KUKA KRL program: dockof_2.src, dockof_2.dat

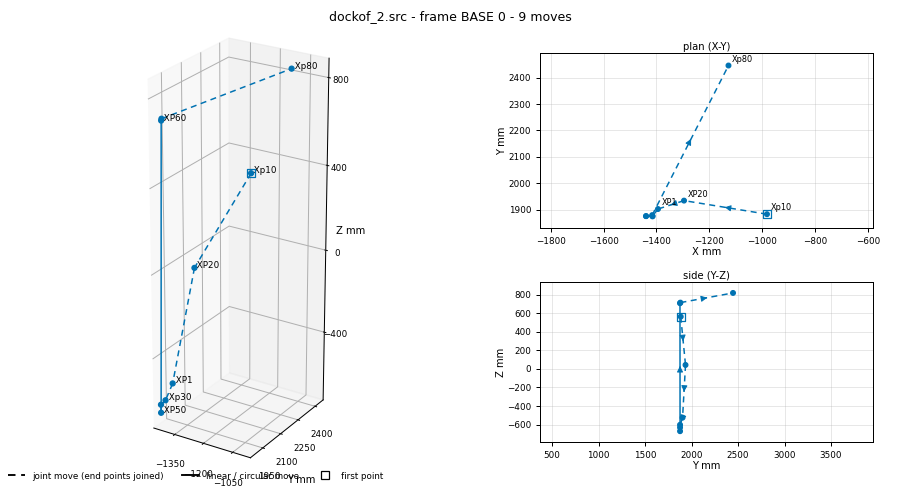
[picture p0: tool path of dockof_2.src in frame BASE 0, 9 of 9 moves have a stored position in this frame; points joined in program order, loops and branches not executed]
--- dockof_2.src ---
&ACCESS RV1
&REL 140
&COMMENT PLACE GUN 2
DEF DOCKOF_2( )
;================================================
; MODEL    :
; IE GROUP :
; STATION  :
; ROBOT    :
; FUNCTION : DOCK OFF GUN 2
;================================================
;FOLD INI
;FOLD BASISTECH INI
GLOBAL INTERRUPT DECL 3 WHEN $STOPMESS==TRUE DO IR_STOPM ( )
INTERRUPT ON 3
BAS (#INITMOV,0 )
;ENDFOLD (BASISTECH INI)
;FOLD GRIPPERTECH INI
USER_GRP(0,DUMMY,DUMMY,GDEFAULT)
;ENDFOLD (GRIPPERTECH INI)
;FOLD USER INI
;Make your modifications here

;ENDFOLD (USER INI)
;ENDFOLD (INI)

;FOLD PTP p10  Vel= 100 % H Tool[2]:Gun2 Base[0];%{PE}%R 5.4.35,%MKUKATPBASIS,%CMOVE,%VPTP,%P 1:PTP, 2:p10, 3:, 5:100, 7:H
$BWDSTART=FALSE
PDAT_ACT=PH
FDAT_ACT=Fp10
BAS(#PTP_PARAMS,100)
PTP Xp10
;ENDFOLD

;Open flap 2
;FOLD DOCKING.FLAP_OPN 2 ;%{PE}%MKUKATPUSER
DOCKING (#FLAP_OPN ,2)
;ENDFOLD

;FOLD ; Check docking station 2 ready to dock off;%{PE}%R 2.4.14,%MKUKATPBASIS,%CCOMMENT,%VNORMAL,%P 2:Check docking station 2 ready to dock off
;ENDFOLD
DOCKING (#REQ_DOCK_OFF ,2)

;FOLD PTP P20 CONT Vel= 100 % h Tool[2]:Gun2 Base[0];%{PE}%R 5.4.35,%MKUKATPBASIS,%CMOVE,%VPTP,%P 1:PTP, 2:P20, 3:C_PTP, 5:100, 7:h
$BWDSTART=FALSE
PDAT_ACT=Ph
FDAT_ACT=FP20
BAS(#PTP_PARAMS,100)
PTP XP20 C_PTP
;ENDFOLD
;FOLD PTP P1 CONT Vel= 100 % H Tool[2]:Gun2 Base[0];%{PE}%R 5.4.35,%MKUKATPBASIS,%CMOVE,%VPTP,%P 1:PTP, 2:P1, 3:C_PTP, 5:100, 7:H
$BWDSTART=FALSE
PDAT_ACT=PH
FDAT_ACT=FP1
BAS(#PTP_PARAMS,100)
PTP XP1 C_PTP
;ENDFOLD
;FOLD PTP p30  Vel= 70 % H Tool[2]:Gun2 Base[0];%{PE}%R 5.4.35,%MKUKATPBASIS,%CMOVE,%VPTP,%P 1:PTP, 2:p30, 3:, 5:70, 7:H
$BWDSTART=FALSE
PDAT_ACT=PH
FDAT_ACT=Fp30
BAS(#PTP_PARAMS,70)
PTP Xp30
;ENDFOLD

;FOLD ; Above dock position station 2;%{PE}%R 2.4.14,%MKUKATPBASIS,%CCOMMENT,%VNORMAL,%P 2:Above dock position station 2
;ENDFOLD
;FOLD PTP p40  Vel= 30 % H Tool[2]:Gun2 Base[0];%{PE}%R 5.4.35,%MKUKATPBASIS,%CMOVE,%VPTP,%P 1:PTP, 2:p40, 3:, 5:30, 7:H
$BWDSTART=FALSE
PDAT_ACT=PH
FDAT_ACT=Fp40
BAS(#PTP_PARAMS,30)
PTP Xp40
;ENDFOLD

;FOLD ; In Dock position Station 2;%{PE}%R 2.4.14,%MKUKATPBASIS,%CCOMMENT,%VNORMAL,%P 2:In Dock position Station 2
;ENDFOLD
;FOLD LIN p50  Vel= 0.2 m/s H Tool[2]:Gun2 Base[0];%{PE}%R 5.4.35,%MKUKATPBASIS,%CMOVE,%VLIN,%P 1:LIN, 2:p50, 3:, 5:0.2, 7:H
$BWDSTART=FALSE
LDAT_ACT=LH
FDAT_ACT=FP50
BAS(#CP_PARAMS,0.2)
LIN XP50
;ENDFOLD

;FOLD ; Unlock Docking plate;%{PE}%R 2.4.14,%MKUKATPBASIS,%CCOMMENT,%VNORMAL,%P 2:Unlock Docking plate
;ENDFOLD
DOCKING (#TOOL_UNLOCK ,2)

;FOLD ; Out Docking station 2;%{PE}%R 2.4.14,%MKUKATPBASIS,%CCOMMENT,%VNORMAL,%P 2:Out Docking station 2
;ENDFOLD
;FOLD LIN p60  Vel= 0.2 m/s H Tool[14]:GRIPPER 1 Base[0];%{PE}%R 5.2.271,%MKUKATPBASIS,%CMOVE,%VLIN,%P 1:LIN, 2:p60, 3:, 5:0.2, 7:H
$BWDSTART = FALSE
LDAT_ACT=LH
FDAT_ACT=FP60
BAS(#CP_PARAMS,0.2)
LIN XP60
;ENDFOLD

;FOLD ; Check docking plate open and station 2 ok;%{PE}%R 2.4.14,%MKUKATPBASIS,%CCOMMENT,%VNORMAL,%P 2:Check docking plate open and station 2 ok
;endfold
DOCKING (#CHK_TOOL_OFF ,2)

;FOLD PTP p70 CONT Vel= 100 % H Tool[10]:Dock plate Base[0];%{PE}%R 5.4.35,%MKUKATPBASIS,%CMOVE,%VPTP,%P 1:PTP, 2:p70, 3:C_PTP, 5:100, 7:H
$BWDSTART=FALSE
PDAT_ACT=PH
FDAT_ACT=Fp70
BAS(#PTP_PARAMS,100)
PTP Xp70 C_PTP
;ENDFOLD
;FOLD PTP p80 CONT Vel= 100 % H Tool[10]:Dock plate Base[0];%{PE}%R 5.4.35,%MKUKATPBASIS,%CMOVE,%VPTP,%P 1:PTP, 2:p80, 3:C_PTP, 5:100, 7:H
$BWDSTART=FALSE
PDAT_ACT=PH
FDAT_ACT=Fp80
BAS(#PTP_PARAMS,100)
PTP Xp80 C_PTP
;ENDFOLD

;Close flap 2
;FOLD DOCKING.FLAP_CLS 2 ;%{PE}%MKUKATPUSER
DOCKING (#FLAP_CLS ,2)
;ENDFOLD
END

--- dockof_2.dat ---
&ACCESS RV1
&REL 140
&COMMENT PLACE GUN 2
DEFDAT  DOCKOF_2
;FOLD EXTERNAL DECLARATIONS;%{PE}%MKUKATPBASIS,%CEXT,%VCOMMON,%P
;FOLD GRIPPERTECH EXT
EXT  H50 (INT  :IN,INT  :IN,INT  :IN,GRP_TYP  :IN )
;ENDFOLD (GRIPPERTECH EXT)
;FOLD SPOTTECH EXT
EXT  USERSPOT (S_COMMAND  :IN,SPOT_TYPE  :IN )
;ENDFOLD (SPOTTECH EXT)
;FOLD BASISTECH EXT;%{PE}%MKUKATPBASIS,%CEXT,%VEXT,%P
EXT  BAS (BAS_COMMAND  :IN,REAL  :IN )
DECL INT SUCCESS
;ENDFOLD (BASISTECH EXT)
;FOLD USER EXT;%{E}%MKUKATPUSER,%CEXT,%VEXT,%P
;Make here your modifications
;ENDFOLD (USER EXT)
;ENDFOLD (EXTERNAL DECLERATIONS)
;*      FDAT Declarations     *

;******************************
;*     E6POS Declarations     *
;******************************

DECL E6POS XP10={X -981.764771,Y 1883.28101,Z 561.632813,A -85.3195038,B 0.149295896,C -0.627375901,S 2,T 43,E1 -735.495178,E2 0.0,E3 0.0,E4 0.0,E5 0.0,E6 0.0}
DECL E6POS XP20={X -1295.61206,Y 1934.646,Z 42.0023003,A -85.3188019,B 0.147270799,C -0.629731119,S 2,T 43,E1 -735.49353,E2 0.0,E3 0.0,E4 0.0,E5 0.0,E6 0.0}
DECL E6POS XP30={X -1415.08899,Y 1875.94202,Z -601.858826,A -85.3188095,B 0.148737103,C -0.630693614,S 2,T 43,E1 -735.491699,E2 0.0,E3 0.0,E4 0.0,E5 0.0,E6 0.0}
DECL E6POS XP40={X -1439.323,Y 1875.89795,Z -630.582214,A -84.2455215,B 0.0450858884,C -0.629668415,S 2,T 43,E1 -735.49353,E2 0.0,E3 0.0,E4 0.0,E5 0.0,E6 0.0}
DECL E6POS XP50={X -1439.32996,Y 1875.90295,Z -670.736511,A -84.2452698,B 0.0452245101,C -0.629822373,S 2,T 43,E1 -735.49353,E2 0.0,E3 0.0,E4 0.0,E5 0.0,E6 0.0}
DECL E6POS XP60={X -1414.71301,Y 1875.07996,Z 706.503113,A -134.240997,B -0.652029216,C 179.492798,S 2,T 43,E1 -735.497009,E2 0.0,E3 0.0,E4 0.0,E5 0.0,E6 0.0}
DECL E6POS XP70={X -1416.05505,Y 1879.71399,Z 712.868896,A -135.317596,B -0.386982203,C 179.484802,S 2,T 43,E1 -735.491699,E2 0.0,E3 0.0,E4 0.0,E5 0.0,E6 0.0}
DECL E6POS XP80={X -1127.36902,Y 2445.76807,Z 816.869385,A -45.7330017,B 0.4947837,C 179.7724,S 2,T 11,E1 -1181.96399,E2 0.0,E3 0.0,E4 0.0,E5 0.0,E6 0.0}

;******************************
;*     FDAT Declarations      *
;******************************

DECL FDAT FP10={TOOL_NO 2,BASE_NO 0,IPO_FRAME #BASE}
DECL FDAT FP20={TOOL_NO 2,BASE_NO 0,IPO_FRAME #BASE}
DECL FDAT FP30={TOOL_NO 2,BASE_NO 0,IPO_FRAME #BASE}
DECL FDAT FP40={TOOL_NO 2,BASE_NO 0,IPO_FRAME #BASE}
DECL FDAT FP50={TOOL_NO 2,BASE_NO 0,IPO_FRAME #BASE}
DECL FDAT FP60={TOOL_NO 14,BASE_NO 0,IPO_FRAME #BASE}
DECL FDAT FP70={TOOL_NO 10,BASE_NO 0,IPO_FRAME #BASE}
DECL FDAT FP80={TOOL_NO 10,BASE_NO 0,IPO_FRAME #BASE}

;******************************
;*  PDAT & LDAT Declarations  *
;******************************

DECL PDAT PH={VEL 100.0,ACC 100.0,APO_DIST 100.0}
DECL LDAT LH={VEL 2.0,ACC 100.0,APO_DIST 100.0,APO_FAC 50.0,ORI_TYP #VAR}

DECL PDAT PPDAT1={VEL 100.0,ACC 100.0,APO_DIST 100.0}
DECL E6POS XP1={X -1394.16199,Y 1902.81897,Z -524.886108,A -85.3188629,B 0.148389801,C -0.63038218,S 2,T 43,E1 -735.491699,E2 0.0,E3 0.0,E4 0.0,E5 0.0,E6 0.0}
DECL FDAT FP1={TOOL_NO 2,BASE_NO 0,IPO_FRAME #BASE,POINT2[] " "}
ENDDAT
